// TIA Portal V17 export
// export: Created 2025-08-05T09:36:01.0887174Z, ExportSetting WithDefaults, DisplayName Totally Integrated Automation Portal, DisplayVersion V17, DisplayName TIA Portal Openness, DisplayVersion V17, DisplayName TIA Portal Version Control Interface, DisplayVersion V17, DisplayName SINAMICS Startdrive Advanced, DisplayVersion V17, DisplayName SINAMICS Startdrive G130, G150, S120, S150, SINAMICS MV, S210, DisplayVersion V17, DisplayName SINAMICS Startdrive G110M, G120, G120C, G120D, G120P, G115D, DisplayVersion V17, DisplayName STEP 7 Professional, DisplayVersion V17, DisplayName STEP 7 Safety, DisplayVersion V17, DisplayName WinCC Advanced, DisplayVersion V17
TYPE "typeMotionOvrvListEntry"
TITLE = Entry motion overview / Eintrag Motion-Übersicht
// Entry motion overview [V 01.00 | Kernel_V2] / Eintrag Motion-Übersicht [V 01.00 | Kernel_V2]
// stored: IsFailsafeCompliant false
   STRUCT
      alive : USInt;   // Alive-Flag (Wird im Motion gesetzt, zentral dann zurückgesetzt) / Alive-Flag (is set in motion, then centrally reset)
      instancePath : String[80];   // Instanzpfad des Motion-Aufrufes (Dient als Identifier) / Instance path of motion call (serves as identifier)
      fgDbAdress : DB_ANY;   // DB-Any Adresse der zugehörigen Funktionsgruppe / DB any address of associated function group
      data : Struct   // Motion-Daten:... / Motion data...
         enable : Bool;   // Grundsätzliche Freigabesignale (Steuerung ein, usw.) / Basic enabling signals (control system on, etc.)
         interlock : Bool;   // Bewegungsverriegelung / Motion interlock
         toPosition : Bool;   // Zur Position aktiv / To position active
         inPosition : Bool;   // In Position / In position
         inPositionStored : Bool;   // Position wurde in Automatik angefahren und wird überwacht / Position was approached in automatic mode and is monitored
         positionValue : LReal;   // Positionswert (optional) / Position value (optional)
         timeOut : Time;   // Überwachungszeit für die Bewegung / Monitoring time for the motion
         timeOfLastMotion : Time;   // Tatsächlich benötigte Zeit der letzten Bewegung / Actually required time of the last motion
      END_STRUCT;
      hmiLine : Struct   // HMI-Zeileninformation / HMI line information
         number : UInt;   // Zeilennummer (0 = keine Zeile) / Line number (0 = no line)
         controSide : SInt;   // Einrichtzeile Links/Rechts (-1 = Links, 0 = keine, 1 = Rechts) / Setup line left/right (-1 = left, 0 = none, 1 = right)
      END_STRUCT;
   END_STRUCT;
END_TYPE
